FUNCTION_BLOCK Station_Core (* Basic Function Block Type *)
  (* Standard: 61499-2 *)
  (* Version 0.0, 7/10/2025, Evans_A, Schneider Electric, Template *)
  PACKAGE Main;
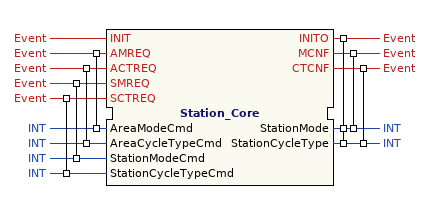
  EVENT_INPUT
    INIT; (* Initialization Request *)
    AMREQ WITH AreaModeCmd; (* Normal Execution Request *)
    ACTREQ WITH AreaCycleTypeCmd;
    SMREQ WITH StationModeCmd;
    SCTREQ WITH StationCycleTypeCmd;
  END_EVENT
  EVENT_OUTPUT
    INITO WITH StationMode, StationCycleType; (* Initialization Confirm *)
    MCNF WITH StationMode; (* Execution Confirmation *)
    CTCNF WITH StationCycleType;
  END_EVENT
  VAR_INPUT
    AreaModeCmd : INT; (* Input event qualifier *)
    AreaCycleTypeCmd : INT;
    StationModeCmd : INT;
    StationCycleTypeCmd : INT;
  END_VAR
  VAR_OUTPUT
    StationMode : INT; (* Output event qualifier *)
    StationCycleType : INT;
  END_VAR
  EC_STATES
    START; (* Initial State *)
    INIT : INIT -> INITO; (* Initialization *)
    AUTO : Auto_Stop -> MCNF, Cycle_Stop -> CTCNF;
    MANUAL : Manual_Stop -> MCNF, Cycle_Stop -> CTCNF;
    SETUP_MODE : Setup_Mode -> MCNF;
    HOME : Initial_Position -> MCNF;
    CONTINUOUS_AUTO : Continuous -> CTCNF;
    STOP_AT_END_AUTO : Stop_At_End -> CTCNF;
    SINGLE_CYCLE_AUTO : Single_Cycle -> CTCNF;
    DRY_CYCLE_AUTO : Dry_Cycle -> CTCNF;
    CONTINUOUS_MANUAL : Continuous -> CTCNF;
    STOP_AT_END_MANUAL : Stop_At_End -> CTCNF;
    SINGLE_CYCLE_MANUAL : Single_Cycle -> CTCNF;
    DRY_CYCLE_MANUAL : Dry_Cycle -> CTCNF;
  END_STATES
  EC_TRANSITIONS
    START TO INIT := INIT;
    INIT TO START := 1;
    START TO AUTO := AMREQ AND AreaModeCmd=1 OR SMREQ AND StationModeCmd=1;
    START TO MANUAL := AMREQ AND AreaModeCmd=2 OR SMREQ AND StationModeCmd=2;
    START TO SETUP_MODE := AMREQ AND AreaModeCmd=3 OR SMREQ AND StationModeCmd=3;
    START TO HOME := AMREQ AND AreaModeCmd=9 OR SMREQ AND StationModeCmd=9;
    AUTO TO MANUAL := AMREQ AND AreaModeCmd=2 OR SMREQ AND StationModeCmd=2;
    MANUAL TO AUTO := AMREQ AND AreaModeCmd=1 OR SMREQ AND StationModeCmd=1;
    AUTO TO SETUP_MODE := AMREQ AND AreaModeCmd=3 OR SMREQ AND StationModeCmd=3;
    SETUP_MODE TO AUTO := AMREQ AND AreaModeCmd=1 OR SMREQ AND StationModeCmd=1;
    AUTO TO HOME := AMREQ AND AreaModeCmd=9 OR SMREQ AND StationModeCmd=9;
    HOME TO AUTO := AMREQ AND AreaModeCmd=1 OR SMREQ AND StationModeCmd=1;
    MANUAL TO SETUP_MODE := AMREQ AND AreaModeCmd=3 OR SMREQ AND StationModeCmd=3;
    SETUP_MODE TO MANUAL := AMREQ AND AreaModeCmd=2 OR SMREQ AND StationModeCmd=2;
    MANUAL TO HOME := AMREQ AND AreaModeCmd=9 OR SMREQ AND StationModeCmd=9;
    HOME TO MANUAL := AMREQ AND AreaModeCmd=2 OR SMREQ AND StationModeCmd=2;
    SETUP_MODE TO HOME := AMREQ AND AreaModeCmd=9 OR SMREQ AND StationModeCmd=9;
    HOME TO SETUP_MODE := AMREQ AND AreaModeCmd=3 OR SMREQ AND StationModeCmd=3;
    AUTO TO CONTINUOUS_AUTO := ACTREQ AND AreaCycleTypeCmd=1 OR SCTREQ AND StationCycleTypeCmd=1;
    AUTO TO STOP_AT_END_AUTO := ACTREQ AND AreaCycleTypeCmd=2 OR SCTREQ AND StationCycleTypeCmd=2;
    AUTO TO SINGLE_CYCLE_AUTO := ACTREQ AND AreaCycleTypeCmd=3 OR SCTREQ AND StationCycleTypeCmd=3;
    SINGLE_CYCLE_AUTO TO AUTO := ACTREQ AND AreaCycleTypeCmd=0 OR SCTREQ AND StationCycleTypeCmd=0;
    STOP_AT_END_AUTO TO AUTO := ACTREQ AND AreaCycleTypeCmd=0 OR SCTREQ AND StationCycleTypeCmd=0;
    CONTINUOUS_AUTO TO AUTO := ACTREQ AND AreaCycleTypeCmd=0 OR SCTREQ AND StationCycleTypeCmd=0;
    AUTO TO DRY_CYCLE_AUTO := ACTREQ AND AreaCycleTypeCmd=4 OR SCTREQ AND StationCycleTypeCmd=4;
    DRY_CYCLE_AUTO TO AUTO := ACTREQ AND AreaCycleTypeCmd=0 OR SCTREQ AND StationCycleTypeCmd=0;
    CONTINUOUS_AUTO TO STOP_AT_END_AUTO := ACTREQ AND AreaCycleTypeCmd=2 OR SCTREQ AND StationCycleTypeCmd=2;
    MANUAL TO CONTINUOUS_MANUAL := ACTREQ AND AreaCycleTypeCmd=1 OR SCTREQ AND StationCycleTypeCmd=1;
    MANUAL TO STOP_AT_END_MANUAL := ACTREQ AND AreaCycleTypeCmd=2 OR SCTREQ AND StationCycleTypeCmd=2;
    CONTINUOUS_MANUAL TO STOP_AT_END_MANUAL := ACTREQ AND AreaCycleTypeCmd=2 OR SCTREQ AND StationCycleTypeCmd=2;
    MANUAL TO SINGLE_CYCLE_MANUAL := ACTREQ AND AreaCycleTypeCmd=3 OR SCTREQ AND StationCycleTypeCmd=3;
    MANUAL TO DRY_CYCLE_MANUAL := ACTREQ AND AreaCycleTypeCmd=4 OR SCTREQ AND StationCycleTypeCmd=4;
    CONTINUOUS_MANUAL TO MANUAL := ACTREQ AND AreaCycleTypeCmd=0 OR SCTREQ AND StationCycleTypeCmd=0;
    STOP_AT_END_MANUAL TO MANUAL := ACTREQ AND AreaCycleTypeCmd=0 OR SCTREQ AND StationCycleTypeCmd=0;
    SINGLE_CYCLE_MANUAL TO MANUAL := ACTREQ AND AreaCycleTypeCmd=0 OR SCTREQ AND StationCycleTypeCmd=0;
    DRY_CYCLE_MANUAL TO MANUAL := ACTREQ AND AreaCycleTypeCmd=0 OR SCTREQ AND StationCycleTypeCmd=0;
  END_TRANSITIONS
  ALGORITHM INIT IN ST: (* Initialization algorithm *)
StationMode := 0;
StationCycleType :=0;
  END_ALGORITHM
  ALGORITHM REQ IN ST: (* Normally executed algorithm *)
;
  END_ALGORITHM
  ALGORITHM Auto_Stop IN ST:
StationMode:=1;
  END_ALGORITHM
  ALGORITHM Manual_Stop IN ST:
StationMode:=2;
  END_ALGORITHM
  ALGORITHM Setup_Mode IN ST:
StationMode:=3;
  END_ALGORITHM
  ALGORITHM Initial_Position IN ST:
StationMode:=9;
  END_ALGORITHM
  ALGORITHM Continuous IN ST:
StationCycleType:=1;
  END_ALGORITHM
  ALGORITHM Stop_At_End IN ST:
StationCycleType:=2;
  END_ALGORITHM
  ALGORITHM Single_Cycle IN ST:
StationCycleType:=3;
  END_ALGORITHM
  ALGORITHM Dry_Cycle IN ST:
StationCycleType:=4;
  END_ALGORITHM
  ALGORITHM Cycle_Stop IN ST:
StationCycleType:=0;
  END_ALGORITHM
END_FUNCTION_BLOCK
